TYPE CM_DIN_UDT :
STRUCT
	SensorInput : BOOL;
	
	AutoHigh : BOOL;
END_STRUCT
END_TYPE

(* stored: Version 1.1.0.1, ProductVersion 3.1.4024.13
   DUT CM_DIN_UDT: Id {19945d24-740f-4b2b-8f70-25667657d4c7} *)
